FUNCTION_BLOCK FB_CartCtrlCycleTest_1 EXTENDS FB_CartCtrlBase
VAR_INPUT
END_VAR
VAR_OUTPUT
END_VAR
VAR
	//左支撑-右支撑-左轮-右轮-立柱升降-横梁旋转-横梁伸缩-悬吊旋转
	//In this method, 5 represents the pillar postion , 6 represents the beam rotation angle ,7 represents the beam stretch position ,8 represents the overhang angle
	
	//test step
	m_testStep:INT:=-1;
	
	//motion start
	m_startMotion:BOOL;
	m_startMotionLast:BOOL;
	
	//time
	m_time:LREAL;
	
	//test point
	//m_testPoint:INT;
	
	//DH joint position	
	m_homeDHJntPos,m_startDHJntPos,m_endDHJntPos:Vec8d;
	
	//startJntPos,endJntPos :Vec8d;
	m_initJntPos,m_startJntPos,m_endJntPos :Vec8d;
	
	//motion distance
	m_motDist:Vec8d;
	
	//cycle time
	m_curCycleTime:LREAL;
	
	//joint position gap
	m_jntDist:Vec8d:=[0,0,0,0,   0.030,30.0*g_deg2Rad,0.030,30.0*g_deg2Rad];	
	
	//planner
	m_Planner: FB_TrajMoveJ;
	
	//trajectory velocity/acceleration/jerk
	m_maxjntVel:Vec8d;
	m_maxjntAcc:Vec8d;
	m_maxjntJerk:Vec8d;
	
	//arm id
	m_armId:INT:=1;
	
	//test point
	m_pointNum:INT;
	
	//point sum
	m_pointSum:INT;
	
	//target cycle number
	m_motionCycleNum:INT;
	m_targetCycleNum:INT;
	
	//target joint position
	m_targetJntPos:ARRAY[1..10] OF Vec8d;
	
	//unit function
	m_unitFun:FB_UnitTransform;
	
	//motion joint velocity limit
	m_motVelLimit:Vec8d:=[0.1,0.1,0.1,0.1,      0.01, 0.02,0.01,0.02];
END_VAR

// override this function in each exact controller
METHOD PROTECTED calcCmdJntPos : BOOL
VAR_IN_OUT CONSTANT
	// slave cart joint data
	i_slaveCart :FB_SlaveCart;
END_VAR

VAR
	i:INT;
END_VAR

//init parameters flag
IF (g_cycleTest.m_carEnterESDTest=TRUE) THEN
	m_startMotion:=TRUE;
ELSE
	m_startMotion:=g_cycleTest.m_startMotionCar;
END_IF

//monitoring signal rising edge
IF (m_startMotionLast=FALSE) AND (m_startMotion=TRUE)THEN
	m_testStep:=0;
END_IF
m_startMotionLast:=m_startMotion;

//frequency test and step test
testMotion(i_slaveCart);

//update the information
updateInfo(i_slaveCart);

//update the information
GVL_Monitor.m_carTargetJntPos:=m_cmdJntPos;
GVL_Monitor.g_carActJntPos:=i_slaveCart.curJntPos;
GVL_Monitor.g_carTestStep:=m_testStep;
GVL_Monitor.g_cartime:=m_time;
END_METHOD

// override this function in each exact controller
// NOTICE: set joint control mode here, and do some initialization if needed
METHOD PUBLIC init : BOOL
VAR_IN_OUT CONSTANT
	i_slaveCart	:FB_SlaveCart;
END_VAR
VAR_IN_OUT 
	r_cartCtrlCmd :ST_SlaveArmCtrlCmds;
END_VAR
VAR
	i:INT;
END_VAR

SUPER^.init(i_slaveCart,r_cartCtrlCmd);

//Drive the last four joints
m_jntEnableFlag :=g_zeroVec8i;
FOR i:=5 TO 8 BY 1 DO
	m_jntEnableFlag[i] :=1;
END_FOR

//operation mode
m_jntOPMode:=g_slaveAllPosMode;
m_jntOPMode[5]:= DriverOPMode_cspMZ;
m_jntOPMode[6]:= DriverOPMode_Pos;
m_jntOPMode[7]:= DriverOPMode_Pos;
m_jntOPMode[8]:= DriverOPMode_Pos;

// update commands to arm
copyCmds(r_cartCtrlCmd);

//target DH joint position
FOR i:=1 TO g_cartJntNum BY 1 DO
	m_homeDHJntPos[i]:=(GVL_CartMotorParameters.g_minJntPos[i]+GVL_CartMotorParameters.g_maxJntPos[i])/2;
	m_jntDist[i]:=(GVL_CartMotorParameters.g_maxJntPos[i]-GVL_CartMotorParameters.g_minJntPos[i])*0.05;
	m_startDHJntPos[i]:=m_homeDHJntPos[i]-m_jntDist[i];
	m_endDHJntPos[i]:=m_homeDHJntPos[i]+m_jntDist[i];
END_FOR

//Keep the first four joints still
FOR i:=1 TO 4 BY 1 DO
	m_homeDHJntPos[i]:=i_slaveCart.curJntPos[i];
	m_startDHJntPos[i]:=m_homeDHJntPos[i];
	m_endDHJntPos[i]:=m_homeDHJntPos[i];
END_FOR

//velocity and acceleration
vecMultiNum(GVL_CartControlParameters.g_maxJntVel,0.1,m_maxjntVel);
vecMultiNum(m_maxjntVel,5,m_maxjntAcc);
vecMultiNum(m_maxjntAcc,5,m_maxjntJerk);

//start flag
m_startMotionLast:=FALSE;

//copy the target joint position value
IF (g_cycleTest.m_carEnterESDTest=FALSE) THEN
	m_pointSum:=g_cycleTest.m_pointSumCar;
	m_targetCycleNum:=g_cycleTest.m_targetCycleNumCar;
	FOR i:=1 TO 10 BY 1 DO
		m_targetJntPos[i]:=m_unitFun.carUnit2System(i_dataTest:= g_cycleTest.m_targetJntPosCar[i]);
	END_FOR	
ELSE
	m_pointSum:=3;
	m_targetCycleNum:=30000;
	m_targetJntPos[1]:=m_startDHJntPos; 	m_targetJntPos[2]:=m_homeDHJntPos;	m_targetJntPos[3]:=m_endDHJntPos;
END_IF
END_METHOD

METHOD testMotion : BOOL
VAR_INPUT
	// slave cart joint data
	i_slaveCart :FB_SlaveCart;
END_VAR
VAR
	homeDHPos,startDHPos,endDHPos :Vec8d;
	i:INT;
END_VAR

CASE m_testStep OF
	0: //init
		IF (g_cycleTest.m_carEnterESDTest=FALSE) THEN
			m_pointSum:=g_cycleTest.m_pointSumCar;
			m_targetCycleNum:=g_cycleTest.m_targetCycleNumCar;
			FOR i:=1 TO 10 BY 1 DO
				m_targetJntPos[i]:=m_unitFun.carUnit2System(i_dataTest:= g_cycleTest.m_targetJntPosCar[i]);
			END_FOR	
		ELSE
			g_cycleTest.m_tgtCycleTimeCar:=1;
			m_pointSum:=3;
			m_targetCycleNum:=30000;
			m_targetJntPos[1]:=m_startDHJntPos; 	m_targetJntPos[2]:=m_homeDHJntPos;	m_targetJntPos[3]:=m_endDHJntPos;
		END_IF
		
		m_maxjntVel:=m_unitFun.carUnit2System(i_dataTest:= g_cycleTest.m_targetJntVelCar);
		FOR i:=1 TO 8 BY 1 DO
			IF ABS(m_maxjntVel[i])<g_smallNum THEN
				m_maxjntVel[i]:=g_cycleTest.m_defultTargetJntVelCar[i];
			END_IF
			m_maxjntVel[i]:=LIMIT(0,m_maxjntVel[i],m_motVelLimit[i]);
		END_FOR
		vecMultiNum(m_maxjntVel,3,m_maxjntAcc);
		vecMultiNum(m_maxjntAcc,3,m_maxjntJerk);	
	
		m_pointNum:=1;
		m_motionCycleNum:=0;
		m_curCycleTime:=0;	
		m_testStep:=10;
		
		
	10: //Trajectory parameter initialization
		startDHPos:=i_slaveCart.curJntPos;
		endDHPos:=m_targetJntPos[m_pointNum];	
		FOR i:=1 TO 4 BY 1 DO
			endDHPos[i]:=startDHPos[i];
		END_FOR		
		
		m_startJntPos:=startDHPos;
		m_endJntPos:=endDHPos;
		
		//limit the joint position
		FOR i:=1 TO 8 BY 1 DO
			m_startJntPos[i]:=LIMIT(GVL_CartMotorParameters.g_minJntPos[i],m_startJntPos[i],GVL_CartMotorParameters.g_maxJntPos[i]);
			m_endJntPos[i]:=LIMIT(GVL_CartMotorParameters.g_minJntPos[i],m_endJntPos[i],GVL_CartMotorParameters.g_maxJntPos[i]);		
		END_FOR
		
		//motion distance judgement
		vecSub(m_endJntPos,m_startJntPos,m_motDist);
		IF (norm(m_motDist)<g_smallNum) THEN
			m_testStep:=25;
			RETURN;
		END_IF
		
		m_Planner.init(i_startJntPos:= m_startJntPos, 	i_targetJntPos:= m_endJntPos, 	i_maxJntVel:= m_maxjntVel, 	i_maxJntAcc:= m_maxjntAcc, 	i_maxJntJerk:= m_maxjntJerk);
		IF (m_Planner.isGene=FALSE) THEN
			m_testStep:=30;
		ELSE
			m_time:=0; m_testStep:=20;
		END_IF
				
	
	20: //start motion
		IF (g_cycleTest.m_pauseCar=TRUE) THEN		
			RETURN;
		END_IF
		
		IF (g_cycleTest.m_finishCar=TRUE) THEN
			g_cycleTest.m_finishCar:=FALSE;
			m_testStep:=30;
			RETURN;
		END_IF	
		
		//end the motion
		IF (m_startMotion=FALSE) THEN
			m_testStep:=30;
		END_IF
						
		//motion duration
		m_time:=m_time+g_setupArmCtrlCycleTime;
		m_Planner.evaluate(t:= m_time, jntPos=> m_cmdJntPos, jntVel=> m_cmdJntVel, jntAcc=> m_cmdJntAcc);		
		IF (m_time>m_Planner.duration) THEN
			m_testStep:=25;
		END_IF		
		
		
	25: //Record the motion cycle
		m_pointNum:=m_pointNum+1;
		IF (m_pointNum>m_pointSum) THEN		
			m_pointNum:=1;
			m_motionCycleNum:=m_motionCycleNum+1;
			//IF (m_motionCycleNum>m_targetCycleNum) THEN
			IF (g_cycleTest.m_curCycleTimeCar>g_cycleTest.m_tgtCycleTimeCar) THEN
				m_testStep:=30;
			ELSE
				m_testStep:=10;
			END_IF
		ELSE
			m_testStep:=10;
		END_IF	
		
		
	30: //end the motion
		m_testStep:=-1;
END_CASE


//time
IF (m_testStep=-1) THEN
	m_curCycleTime:=0;
ELSE
	m_curCycleTime:=m_curCycleTime+g_cartCtrlCycleTime;
END_IF
g_cycleTest.m_curCycleTimeCar:=m_curCycleTime/3600;


//feedback the information to ui
g_cycleTest.m_curPointNumCar:=m_pointNum;
g_cycleTest.m_curCycleNumCar:=m_motionCycleNum;
g_cycleTest.m_stepNumCar:=m_testStep;
END_METHOD

METHOD updateInfo : BOOL
VAR_INPUT
	// slave cart joint data
	i_slaveCart :FB_SlaveCart;
END_VAR
VAR
	i:INT;
END_VAR

FOR i:=1 TO g_cartJntNum BY 1 DO
	g_cycleTest.m_cartMotorEncoder[i]:=i_slaveCart.m_cartJoints[i].m_motorInputs.m_motorEncoder;
	g_cycleTest.m_cartjntEncoder[i]:=i_slaveCart.m_cartJoints[i].m_motorInputs.m_linkEncoder;
END_FOR

//current joint position
g_cycleTest.m_actJntPosCar:=m_unitFun.carArmUnit2User(i_dataSystem:= i_slaveCart.curJntPos);

//cover the target joint position
IF (g_cycleTest.m_coverCmdPosCar=TRUE) THEN
	i:=g_cycleTest.m_pntIdForCoverCmdCar;
	IF (i>=1) AND (i<=10) THEN
		g_cycleTest.m_targetJntPosCar[i]:=m_unitFun.carArmUnit2User(i_dataSystem:= i_slaveCart.curJntPos);
		m_targetJntPos[i]:=i_slaveCart.curJntPos;
	END_IF
END_IF
END_METHOD

END_FUNCTION_BLOCK

(* stored: Version 1.1.0.1, ProductVersion 3.1.4024.11
   POU FB_CartCtrlCycleTest_1: Id {d1137cb7-190a-40de-acd2-b60cdc071d70}, SpecialFunc None
   Method calcCmdJntPos: Id {19dc3c3d-ae60-4c16-b841-972160fa205a}
   Method init: Id {afe2bec9-2d87-4a06-9c07-4b913474121a}
   Method testMotion: Id {30a813f2-17d5-484f-88cf-325fb776d10a}
   Method updateInfo: Id {64ef6ad7-c09d-4da9-9ca1-550c3567e6cd} *)
